FUNCTION_BLOCK PUBLIC Recipe2
VAR_INPUT
	ExecutingRecipe2: BOOL;
END_VAR
VAR_OUTPUT
	SuccesfullyEnded: BOOL := FALSE;
END_VAR
VAR
	State: INT := 0;
	InitialRotationPosition: INT := 140;
	InitialLiftingPosition: INT := 200;
	MaxGripPosition: INT := 160;
END_VAR

// Recipe is sequence of moves to execute the task.

IF ExecutingRecipe2 THEN	// we start executing recipe2 (again)
	SuccesfullyEnded := FALSE;
END_IF

IF NOT IO.Switch AND NOT SuccesfullyEnded THEN
	// WOOD:
	IF State = 0 THEN
		IF Automatic.RotationPositionAuto < InitialRotationPosition THEN
			IO.MotorRotationDirection := 0;
			IF NOT Automatic.SafetyRON THEN
				Automatic.RCurrentlyMoving := TRUE;
				IO.MotorRotation := 1;
			END_IF
		ELSE
			State := 1;
			IO.MotorRotation := 0;
			Automatic.RCurrentlyMoving := FALSE;
		END_IF
	ELSIF State = 1 THEN
		IF Automatic.LiftingPositionAuto < InitialLiftingPosition THEN
			IO.MotorLiftingDirection := 1;
			IF NOT Automatic.SafetyLON THEN
				Automatic.LCurrentlyMoving := TRUE;
				IO.MotorLifting := 1;
			END_IF
		ELSE
			State := 2;
			IO.MotorLifting := 0;
			Automatic.LCurrentlyMoving := FALSE;
		END_IF
	ELSIF State = 2 THEN
		IF Automatic.GripPositionAuto < MaxGripPosition THEN
			IO.MotorGripDirection := 0;
			IF NOT Automatic.SafetyGON THEN
				Automatic.GCurrentlyMoving := TRUE;
				IO.MotorGrip := 1;
			END_IF
		ELSE
			State := 3;
			IO.MotorGrip := 0;
			Automatic.GCurrentlyMoving := FALSE;
		END_IF
	ELSIF State = 3 THEN
		IF NOT IO.EndLiftingSensor THEN
			IO.MotorLiftingDirection := 0;
			IF NOT Automatic.SafetyLON THEN
				Automatic.GCurrentlyMoving := TRUE;
				IO.MotorLifting := 1;
			END_IF
		ELSE
			State := 4;
			IO.MotorLifting := 0;
			Automatic.GCurrentlyMoving := FALSE;
		END_IF
	ELSIF State = 4 THEN
		IF NOT IO.EndRotationSensor THEN
			IO.MotorRotationDirection := 1;
			IF NOT Automatic.SafetyRON THEN
				Automatic.RCurrentlyMoving := TRUE;
				IO.MotorRotation := 1;
			END_IF
		ELSE
			State := 5;
			IO.MotorRotation := 0;
			Automatic.RCurrentlyMoving := FALSE;
		END_IF
	ELSIF State = 5 THEN
		IF NOT IO.EndGripSensor THEN		// it places the cylinder onto the platform
			IO.MotorGripDirection := 1;
			IF NOT Automatic.SafetyGON THEN
				Automatic.GCurrentlyMoving := TRUE;
				IO.MotorGrip := 1;
			END_IF
		ELSE
			State := 6;
			IO.MotorGrip := 0;
			Automatic.GCurrentlyMoving := FALSE;
		END_IF
	ELSIF State = 6 THEN
		SuccesfullyEnded := TRUE;
		State := 0;
		RETURN;
	END_IF
END_IF

END_FUNCTION_BLOCK

(* stored: Version 1.1.0.1, ProductVersion 3.1.4024.13
   POU Recipe2: Id {cefbc20c-159f-4896-912e-87a831f8ea44}, SpecialFunc None *)
